// Implicitly generated code : DO NOT EDIT
FUNCTION CheckDivLInt : LINT
VAR_INPUT
	divisor:LINT;
END_VAR

// Implicitly generated code : Only an Implementation suggestion
{noflow}
IF divisor = 0 THEN
	CheckDivLInt:=1;
		divisionCheckCounter:= divisionCheckCounter + 1;

ELSE
	CheckDivLInt:=divisor;
END_IF;
{flow}

END_FUNCTION

(* stored: Version 1.1.0.1, ProductVersion 3.1.4024.15
   POU CheckDivLInt: Id {b0cb745d-0312-4472-9e8c-dc4f6bea233a}, SpecialFunc CheckDivInt64 *)
